PROGRAM main
VAR
	Start AT %QX0.0 : bool;
	StopCircuitHealthy AT %QX0.1 : bool;
	SystemActive AT %QX0.2 : bool;
END_VAR

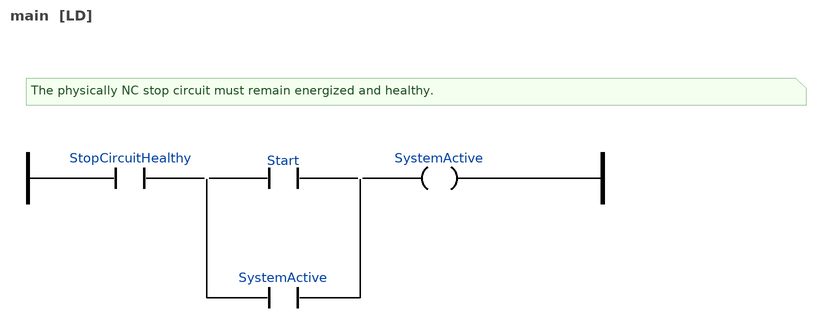
(* LD diagram, written out as Structured Text *)
(* The physically NC stop circuit must remain energized and healthy. *)
SystemActive := StopCircuitHealthy AND (Start OR SystemActive);
END_PROGRAM
